FUNCTION_BLOCK FB_VICI_EPS_TEST EXTENDS FB_TestSuite
VAR_INPUT
END_VAR
VAR_OUTPUT
END_VAR
VAR

END_VAR

TestRequestEpsNotOkPortExpectNoPortChange();
TestActivePortBecomesLockedExpectExternalSignalSetTrue();
TestAllPortsLockedExpectbAllPortsLockedToBeTrue();
TestEpsPortStatusChangeExpectPortStatusToChange();
TestLockedPortMovesWithOverrideExpectPortToMove();

METHOD TestActivePortBecomesLockedExpectExternalSignalSetTrue :  REFERENCE TO FB_Test
VAR
	fbViciEPS : FB_4PVICI_EPS;
	aEPS : ARRAY[1..4] OF DUT_VICI_PORT_EPS;
	
	fbEPS : FB_EPS;
	
	bAllPortsLocked : BOOL;
	bExternalSignal : BOOL;
	iReqNewPort : INT;	
END_VAR
TEST('TestActivePortBecomesLockedExpectExternalSignalSetTrue');
fbEPS(eps:=aEPS[1].stEPS);
fbEPS.setBit(0, TRUE);

fbEPS(eps:=aEPS[2].stEPS);
fbEPS.setBit(0, TRUE);

fbEPS(eps:=aEPS[3].stEPS);
fbEPS.setBit(0, TRUE);

fbEPS(eps:=aEPS[4].stEPS);
fbEPS.setBit(0, TRUE);

iReqNewPort := fbViciEPS.M_EPS_LOGIC(
	aPortEPS := aEPS, 
	iReqPort := 1 ,
	iPrevPort := iReqNewPort,
	bOverride := FALSE,
	bExternalLockSignal => bExternalSignal,
	bAllPortsLocked => bAllPortsLocked
);

AssertEquals_BOOL(
	Expected:= FALSE ,
	Actual:= bExternalSignal,
    Message:= 'bExternalSignal Should be FALSE'
);

fbEPS(eps:=aEPS[1].stEPS);
fbEPS.setBit(0, FALSE);

fbEPS(eps:=aEPS[2].stEPS);
fbEPS.setBit(0, TRUE);

fbEPS(eps:=aEPS[3].stEPS);
fbEPS.setBit(0, TRUE);

fbEPS(eps:=aEPS[4].stEPS);
fbEPS.setBit(0, TRUE);

iReqNewPort := fbViciEPS.M_EPS_LOGIC(
	aPortEPS := aEPS, 
	iReqPort := 1 ,
	iPrevPort := iReqNewPort,
	bOverride := FALSE,
	bExternalLockSignal => bExternalSignal,
	bAllPortsLocked => bAllPortsLocked
);

AssertEquals_BOOL(
	Expected:= TRUE ,
	Actual:= bExternalSignal,
    Message:= 'bExternalSignal Should be TRUE'
);

// CHECK OVERRIDE

iReqNewPort := fbViciEPS.M_EPS_LOGIC(
	aPortEPS := aEPS, 
	iReqPort := 1 ,
	iPrevPort := iReqNewPort,
	bOverride := TRUE,
	bExternalLockSignal => bExternalSignal,
	bAllPortsLocked => bAllPortsLocked
);

AssertEquals_BOOL(
	Expected:= FALSE ,
	Actual:= bExternalSignal,
    Message:= 'bExternalSignal Should be FALSE'
);

TEST_FINISHED();
END_METHOD

METHOD TestAllPortsLockedExpectbAllPortsLockedToBeTrue :  REFERENCE TO FB_Test
VAR_INPUT
END_VAR
VAR
	fbViciEPS : FB_4PVICI_EPS;
	aEPS : ARRAY[1..4] OF DUT_VICI_PORT_EPS;
	
	fbEPS : FB_EPS;
	
	bAllPortsLocked : BOOL;
	iReqNewPort : INT;	
END_VAR
TEST('TestAllPortsLockedExpectbAllPortsLockedToBeTrue');
fbEPS(eps:=aEPS[1].stEPS);
fbEPS.setBit(0, TRUE);

fbEPS(eps:=aEPS[2].stEPS);
fbEPS.setBit(0, TRUE);

fbEPS(eps:=aEPS[3].stEPS);
fbEPS.setBit(0, TRUE);

fbEPS(eps:=aEPS[4].stEPS);
fbEPS.setBit(0, TRUE);

iReqNewPort := fbViciEPS.M_EPS_LOGIC(
	aPortEPS := aEPS, 
	iReqPort := 1 ,
	iPrevPort := iReqNewPort,
	bOverride := FALSE,
	bAllPortsLocked => bAllPortsLocked
);

AssertEquals_BOOL(
	Expected:= FALSE ,
	Actual:= bAllPortsLocked,
    Message:= 'ALL PORTS ARE LOCKED'
);

fbEPS(eps:=aEPS[1].stEPS);
fbEPS.setBit(0, FALSE);

fbEPS(eps:=aEPS[2].stEPS);
fbEPS.setBit(0, FALSE);

fbEPS(eps:=aEPS[3].stEPS);
fbEPS.setBit(0, FALSE);

fbEPS(eps:=aEPS[4].stEPS);
fbEPS.setBit(0, FALSE);

iReqNewPort := fbViciEPS.M_EPS_LOGIC(
	aPortEPS := aEPS, 
	iReqPort := 1 ,
	bOverride := FALSE,
	iPrevPort := iReqNewPort,
	bAllPortsLocked => bAllPortsLocked
);

AssertEquals_BOOL(
	Expected:= TRUE ,
	Actual:= bAllPortsLocked,
    Message:= 'ALL PORTS ARE NOT LOCKED'
);

TEST_FINISHED();
END_METHOD

METHOD TestEpsPortStatusChangeExpectPortStatusToChange :  REFERENCE TO FB_Test
VAR_INPUT
END_VAR
VAR
	fbViciEPS : FB_4PVICI_EPS;
	aEPS : ARRAY[1..4] OF DUT_VICI_PORT_EPS;
	
	fbEPS : FB_EPS;
	
	bAllPortsLocked : BOOL;
	iReqNewPort : INT;
END_VAR
TEST('TestEpsPortStatusChangeExpectPortStatusToChange');
fbEPS(eps:=aEPS[1].stEPS);
fbEPS.setBit(0, TRUE);

fbEPS(eps:=aEPS[2].stEPS);
fbEPS.setBit(0, TRUE);

fbEPS(eps:=aEPS[3].stEPS);
fbEPS.setBit(0, TRUE);

fbEPS(eps:=aEPS[4].stEPS);
fbEPS.setBit(0, TRUE);

// MAKE PORT 1 ACTIVE
iReqNewPort := fbViciEPS.M_EPS_LOGIC(
	aPortEPS := aEPS, 
	iReqPort := 1 ,
	iPrevPort := iReqNewPort,
	bOverride := FALSE,
	bAllPortsLocked => bAllPortsLocked
);

AssertEquals_INT(
	Expected:= ENUM_PORT_STATUS.ACTIVE ,
	Actual:= aEPS[1].ePortStatus,
    Message:= 'PORT 1: NOT ACTIVE'
);

// MAKE PORT 1 UNLOCKED 
iReqNewPort := fbViciEPS.M_EPS_LOGIC(
	aPortEPS := aEPS, 
	iReqPort := 2 ,
	iPrevPort := iReqNewPort,
	bOverride := FALSE,
	bAllPortsLocked => bAllPortsLocked
);

AssertEquals_INT(
	Expected:= ENUM_PORT_STATUS.UNLOCKED ,
	Actual:= aEPS[1].ePortStatus,
    Message:= 'PORT 1: NOT IN UNLOCKED STATE'
);

// MAKE PORT 1 LOCKED
fbEPS(eps:=aEPS[1].stEPS);
fbEPS.setBit(0, FALSE);

iReqNewPort := fbViciEPS.M_EPS_LOGIC(
	aPortEPS := aEPS, 
	iReqPort := 2 ,
	iPrevPort := iReqNewPort,
	bOverride := FALSE,
	bAllPortsLocked => bAllPortsLocked
);

AssertEquals_INT(
	Expected:= ENUM_PORT_STATUS.LOCKED ,
	Actual:= aEPS[1].ePortStatus,
    Message:= 'PORT 1: NOT IN LOCKED STATE'
);

TEST_FINISHED();
END_METHOD

METHOD TestLockedPortMovesWithOverrideExpectPortToMove :  REFERENCE TO FB_Test
VAR_INPUT
END_VAR
VAR
	fbViciEPS : FB_4PVICI_EPS;
	aEPS : ARRAY[1..4] OF DUT_VICI_PORT_EPS;
	
	fbEPS : FB_EPS;
	bAllPortsLocked : BOOL;
	iReqNewPort : INT;
END_VAR
TEST('TestLockedPortMovesWithOverrideExpectPortToMove');
fbEPS(eps:=aEPS[1].stEPS);
fbEPS.setBit(0, TRUE);

fbEPS(eps:=aEPS[2].stEPS);
fbEPS.setBit(0, TRUE);

fbEPS(eps:=aEPS[3].stEPS);
fbEPS.setBit(0, FALSE);

fbEPS(eps:=aEPS[4].stEPS);
fbEPS.setBit(0, TRUE);

// REQUEST PORT 1
iReqNewPort := fbViciEPS.M_EPS_LOGIC(aPortEPS := aEPS, 
	iReqPort := 1 ,
	iPrevPort := iReqNewPort,
	bOverride := FALSE,
	bAllPortsLocked => bAllPortsLocked);

AssertEquals_INT(Expected:= 1 ,
	Actual:= iReqNewPort,
    Message:= 'VICI EPS DID NOT MOVE TO ALLOWED PORT');

// REQUEST PORT 3
iReqNewPort := fbViciEPS.M_EPS_LOGIC(aPortEPS := aEPS, 
	iReqPort := 3 ,
	iPrevPort := iReqNewPort,
	bOverride := TRUE, // OVERRIDE ENABLED
	bAllPortsLocked => bAllPortsLocked);

AssertEquals_INT(Expected:= 3 ,
	Actual:= iReqNewPort,
    Message:= 'VICI EPS OVERRIDE FAILED');
	
TEST_FINISHED();
END_METHOD

METHOD TestRequestEpsNotOkPortExpectNoPortChange :  REFERENCE TO FB_Test
VAR_INPUT
END_VAR
VAR
	fbViciEPS : FB_4PVICI_EPS;
	aEPS : ARRAY[1..4] OF DUT_VICI_PORT_EPS;
	fbEPS : FB_EPS;
	bAllPortsLocked : BOOL;
	iReqNewPort : INT;
END_VAR
TEST('TestRequestEpsNotOkPortExpectNoPortChange');

fbEPS(eps:=aEPS[1].stEPS);
fbEPS.setBit(0, TRUE);

fbEPS(eps:=aEPS[2].stEPS);
fbEPS.setBit(0, TRUE);

fbEPS(eps:=aEPS[3].stEPS);
fbEPS.setBit(0, FALSE);

fbEPS(eps:=aEPS[4].stEPS);
fbEPS.setBit(0, TRUE);

// REQUEST PORT 1
iReqNewPort := fbViciEPS.M_EPS_LOGIC(aPortEPS := aEPS, 
	iReqPort := 1 ,
	iPrevPort := iReqNewPort,
	bOverride := FALSE,
	bAllPortsLocked => bAllPortsLocked);

AssertEquals_INT(Expected:= 1 ,
	Actual:= iReqNewPort,
    Message:= 'VICI EPS DID NOT MOVE TO ALLOWED PORT');

// REQUEST PORT 3
iReqNewPort := fbViciEPS.M_EPS_LOGIC(aPortEPS := aEPS, 
	iReqPort := 3 ,
	iPrevPort := iReqNewPort,
	bOverride := FALSE,
	bAllPortsLocked => bAllPortsLocked);

AssertEquals_INT(Expected:= 1 ,
	Actual:= iReqNewPort,
    Message:= 'VICI EPS MOVED TO BLOCKED PORT');
	
	
TEST_FINISHED();
END_METHOD

END_FUNCTION_BLOCK

(* stored: Version 1.1.0.1, ProductVersion 3.1.4024.12
   POU FB_VICI_EPS_TEST: Id {9e7a45ca-c992-443a-af30-6d6586b9a3e1}, SpecialFunc None
   Method TestActivePortBecomesLockedExpectExternalSignalSetTrue: Id {410125a3-8cc0-4ee9-90f5-443f51d6ea3e}
   Method TestAllPortsLockedExpectbAllPortsLockedToBeTrue: Id {d7534117-3ba8-42eb-8609-ee403d58a03b}
   Method TestEpsPortStatusChangeExpectPortStatusToChange: Id {89ca8612-4d1a-4a67-a4ac-7c1f417d6511}
   Method TestLockedPortMovesWithOverrideExpectPortToMove: Id {6a29d7d9-78d4-48e7-80e2-1bedbd3bcb74}
   Method TestRequestEpsNotOkPortExpectNoPortChange: Id {2deb68af-d1f2-4ae5-8783-ea2517fe3682} *)
